FUNCTION_BLOCK Referenzfahrt
VAR_INPUT
	//Taster
	Kein_Notaus : BOOL;
	Programm_Einzelsatz : BOOL;
	Zyklus_Start : BOOL;
	Zyklus_Stopp : BOOL;
	//Merker
	SFCInit : BOOL;
	SFCTip : BOOL;
	SFCTipMode : BOOL;
	//Sensoren	
	Endl_Saege_Oben : BOOL;
	Endl_Obere_Stammklemmung_Oben : BOOL;
	Endl_Untere_Stammklemmung_Unten : BOOL;
	Endl_Zufuehrer_Hinten : BOOL;
	
END_VAR
VAR_OUTPUT
	Saege_Heben : BOOL;
	Stammklemmung_oben_Hoch : BOOL;
	Stammklemmung_unten_Runter : BOOL;
	Zufuehrer_Zurueck : BOOL;
	Warten_Auf_Weiterschalten : BOOL;
	QHydraulik_EIN : BOOL;

END_VAR
VAR_IN_OUT
	//Merker
	busy : BOOL;
	
	Referenz_Gefahren : BOOL;
	Zyklus_Beendet : BOOL;
	
END_VAR
VAR
END_VAR

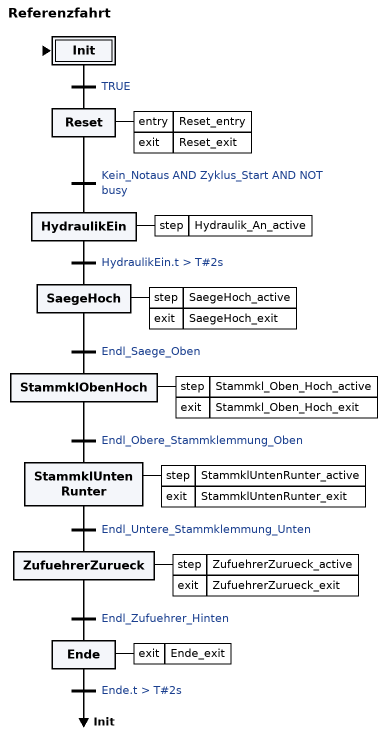
INITIAL_STEP Init:
END_STEP
TRANSITION FROM Init TO Reset
    := TRUE;
END_TRANSITION
STEP Reset:
    Reset_entry(P1);  // entry action
    Reset_exit(P0);  // exit action
END_STEP
TRANSITION FROM Reset TO HydraulikEin
    := Kein_Notaus AND Zyklus_Start AND NOT busy;
END_TRANSITION
STEP HydraulikEin:
    Hydraulik_An_active(N);  // step action
END_STEP
TRANSITION FROM HydraulikEin TO SaegeHoch
    := HydraulikEin.t > T#2s;
END_TRANSITION
STEP SaegeHoch:
    SaegeHoch_active(N);  // step action
    SaegeHoch_exit(P0);  // exit action
END_STEP
TRANSITION FROM SaegeHoch TO StammklObenHoch
    := Endl_Saege_Oben;
END_TRANSITION
STEP StammklObenHoch:
    Stammkl_Oben_Hoch_active(N);  // step action
    Stammkl_Oben_Hoch_exit(P0);  // exit action
END_STEP
TRANSITION FROM StammklObenHoch TO StammklUntenRunter
    := Endl_Obere_Stammklemmung_Oben;
END_TRANSITION
STEP StammklUntenRunter:
    StammklUntenRunter_active(N);  // step action
    StammklUntenRunter_exit(P0);  // exit action
END_STEP
TRANSITION FROM StammklUntenRunter TO ZufuehrerZurueck
    := Endl_Untere_Stammklemmung_Unten;
END_TRANSITION
STEP ZufuehrerZurueck:
    ZufuehrerZurueck_active(N);  // step action
    ZufuehrerZurueck_exit(P0);  // exit action
END_STEP
TRANSITION FROM ZufuehrerZurueck TO Ende
    := Endl_Zufuehrer_Hinten;
END_TRANSITION
STEP Ende:
    Ende_exit(P0);  // exit action
END_STEP
TRANSITION FROM Ende TO Init
    := Ende.t > T#2s;
END_TRANSITION

ACTION Abschluss_active:

END_ACTION

ACTION Ende_exit:
QHydraulik_EIN := FALSE;

busy := FALSE;
Referenz_Gefahren := TRUE;
Zyklus_Beendet := TRUE;
END_ACTION

ACTION Hydraulik_An_active:
QHydraulik_EIN := TRUE;

IF Kein_Notaus AND Zyklus_Start AND NOT busy AND Programm_Einzelsatz THEN 
	Warten_Auf_Weiterschalten := TRUE;
END_IF
END_ACTION

ACTION Hydraulik_An_exit:

END_ACTION

ACTION Reset_entry:
busy := FALSE;
QHydraulik_EIN := FALSE;
Saege_Heben := FALSE;
Stammklemmung_oben_Hoch := FALSE;
Stammklemmung_unten_Runter := FALSE;
Zufuehrer_Zurueck := FALSE;
END_ACTION

ACTION Reset_exit:
busy := TRUE;
Referenz_Gefahren := FALSE;
Zyklus_Beendet := FALSE;

Saege_Heben := FALSE;
Stammklemmung_oben_Hoch := FALSE;
Stammklemmung_unten_Runter := FALSE;
Zufuehrer_Zurueck := FALSE;
END_ACTION

ACTION SaegeHoch_active:
IF NOT Endl_Saege_Oben THEN
	Saege_Heben := TRUE;
END_IF
END_ACTION

ACTION SaegeHoch_exit:
Saege_Heben := FALSE;
END_ACTION

ACTION Stammkl_Oben_Hoch_active:
IF NOT Endl_Obere_Stammklemmung_Oben THEN
	Stammklemmung_oben_Hoch := TRUE;
END_IF
END_ACTION

ACTION Stammkl_Oben_Hoch_exit:
Stammklemmung_oben_Hoch := FALSE;
END_ACTION

ACTION StammklUntenRunter_active:
IF NOT Endl_Untere_Stammklemmung_Unten THEN
	Stammklemmung_unten_Runter := TRUE;
END_IF
END_ACTION

ACTION StammklUntenRunter_exit:
Stammklemmung_unten_Runter := False;
END_ACTION

ACTION ZufuehrerZurueck_active:
IF NOT Endl_Zufuehrer_Hinten THEN
	Zufuehrer_Zurueck := TRUE;
END_IF
END_ACTION

ACTION ZufuehrerZurueck_exit:
Zufuehrer_Zurueck := FALSE;
END_ACTION

END_FUNCTION_BLOCK

(* stored: Version 1.1.0.1, ProductVersion 3.1.4024.16
   POU Referenzfahrt: Id {9a52b441-711b-460e-af45-a6bf65171e00}, SpecialFunc None
   Action Abschluss_active: Id {73c6b22b-fa1f-4b49-969d-aaf633681f09}
   Action Ende_exit: Id {1672a3e4-67b0-4be6-bc60-cb8cfe2f5b24}
   Action Hydraulik_An_active: Id {7246612a-4487-4a08-a6b6-376711e720c2}
   Action Hydraulik_An_exit: Id {31f64795-c125-4cb1-8e29-4526fbdc7e2f}
   Action Reset_entry: Id {6012bee7-c849-43f8-aa0b-86f30e27c83a}
   Action Reset_exit: Id {9ab3edb1-63b0-4841-8792-bcba287ba3d2}
   Action SaegeHoch_active: Id {fb0fbd67-0b64-45fc-91b0-7e6e3da61cdd}
   Action SaegeHoch_exit: Id {8f298d13-0154-419e-a28e-4978d99f6581}
   Action Stammkl_Oben_Hoch_active: Id {e80862e7-3f6b-4e1a-a4a7-4c9b44becc0a}
   Action Stammkl_Oben_Hoch_exit: Id {2df2d016-c626-421e-95c9-201f1305f0a6}
   Action StammklUntenRunter_active: Id {c2b9c445-1400-4bac-9d5f-bf96125c8de0}
   Action StammklUntenRunter_exit: Id {fb3dac32-aa8c-4383-ad20-6c543564ec2c}
   Action ZufuehrerZurueck_active: Id {032bc72d-2cab-4a9c-bdb5-ddb2f3f995fd}
   Action ZufuehrerZurueck_exit: Id {041e648c-93a6-42a9-bdee-1ade29165d0e} *)
